(* CoDeSys 2.3 export: DISCRETESENSCLASS.EXP *)

(* Data type in ENUM *)
TYPE DiscreteSensClass : (DiscreteIn:=1, Counter);
END_TYPE
